//---------------------------------------------------------------------------------------------------------------
//
//  fb_Configuration
//
//  HAUD 2023.04.14
//  - base xml integration
//
//  HAUD 2026.04.10.
//  - now extending a base class
//
//  - cyclic OnChange wrapper for xml data 
//      - Ctrl/State
//        1. INIT
//        2. READ / WRITE
//
//  - read  ST_STATION_PARAMETER on demand
//  - write ST_STATION_PARAMETER on demand
//
//---------------------------------------------------------------------------------------------------------------
// This SOFTWARE is provided as an Example by THE PROVIDER "as is" and "with all faults." THE PROVIDER makes no 
// representations or warranties of any kind concerning the safety, suitability, lack of viruses, inaccuracies, 
// typographical errors, or other harmful components of this SOFTWARE. There are inherent dangers in the use of 
// any software, and you are solely responsible for determining whether this SOFTWARE is compatible with your 
// equipment and other software installed on your equipment. You are also solely responsible for the protection 
// of your equipment and backup of your data, and THE PROVIDER will not be liable for any damages you may suffer 
// in connection with using, modifying, or distributing this SOFTWARE.
//---------------------------------------------------------------------------------------------------------------
FUNCTION_BLOCK fb_Configuration EXTENDS fb_XmlBase
VAR
  _stCtrl               : REFERENCE TO ST_DATA_CTRL;
  _stState              : REFERENCE TO ST_DATA_STATE;

  _stConfiguration      : ST_Configuration;
  _pParameter           : POINTER TO ST_CONFIG_PORTAL;
END_VAR
VAR CONSTANT
  FILE_ROOT             : STRING := 'CONFIG_APPLICATION_';
  X_PATH                : STRING := '/config';
END_VAR

//---------------------------------------------------------------------------------------------------------------
//  check pointers from the outside
//---------------------------------------------------------------------------------------------------------------
IF NOT Check() THEN RETURN; END_IF
//---------------------------------------------------------------------------------------------------------------
// always build the internal data pointer
//  - as always: better safe than sorry
//  - leave this bit here, it doesn't cost much and safely addresses the data
//---------------------------------------------------------------------------------------------------------------
_pData                        := ADR    (_stConfiguration);
_nData                        := SIZEOF (_stConfiguration);
_sXpath                       := X_PATH;

// copy to local for debug
_eCmd                         := _stCtrl.Cmd;

// cyclic check for command change
// get state for cmd
IF (_eCmd <> _eCmdOld)
THEN
  // get matching sdtate for Ctrl.Cmd
  _eState                     := Cmd(_eCmd);
  _eCmdOld                    := _eCmd;
END_IF


CASE _eResult
OF
  E_PROGRESS.PROGRESS_INVALID:
    _stState.State            := E_DATA_STATE.NULL;

  E_PROGRESS.PROGRESS_ERROR:
    _stState.State            := _eState + E_PROGRESS.PROGRESS_ERROR;

  E_PROGRESS.PROGRESS_DONE:
    _stState.State            := _eState + E_PROGRESS.PROGRESS_DONE;

ELSE
  // work in progress
  // update progress for extern use
  _stState.State              := _eState + _eResult;

  CASE _eState
  OF
    E_DATA_STATE.INIT:
      _eResult   := _eInit    := CreateFolder(TRUE);

    E_DATA_STATE.READ:
      _eResult                := XmlRead(TRUE);
      IF (_eResult = E_PROGRESS.PROGRESS_DONE)
      THEN
        // copy the single ladies
        memcpy(_pParameter, ADR(_stConfiguration.PortalConfig), SIZEOF(_stConfiguration.PortalConfig));
      END_IF

    E_DATA_STATE.WRITE:
      _eResult                := XmlWrite(TRUE);
  ELSE
      _eResult                := E_PROGRESS.PROGRESS_INVALID;
  END_CASE
END_CASE

METHOD Check : BOOL
//-------------------------------------------------------------------------
IF NOT (__ISVALIDREF(_stCtrl))
THEN
  _eCheck               := E_DATA_CHECK.REFERENCE_CTRL_INVALID;
  RETURN;
END_IF
//-------------------------------------------------------------------------
IF NOT (__ISVALIDREF(_stState))
THEN
  _eCheck               := E_DATA_CHECK.REFERENCE_STATE_INVALID;
  RETURN;
END_IF
//-------------------------------------------------------------------------
IF NOT (_pStationParameter <> 0)
THEN
  _eCheck               := E_DATA_CHECK.POINTER_STATION_PARAMETER_INVALID;
  RETURN;
END_IF
//-------------------------------------------------------------------------
_eCheck                 := E_DATA_CHECK.DONE_CHECK;
Check                   := TRUE;
END_METHOD

METHOD PRIVATE Cmd : E_DATA_STATE
VAR_INPUT
  Ctrl      : E_DATA_CTRL;
END_VAR
VAR_INST
  _eState   : E_DATA_STATE;
END_VAR
IF NOT Check() THEN Cmd   := E_DATA_STATE.NULL;  RETURN; END_IF

CASE Ctrl
OF
  //---------------------------------------------------------------
  E_DATA_CTRL.INIT:
    _sName                := concat(FILE_ROOT, _sIdentity);
    _sName                := concat(_sName, '.xml');
    _sFilePath            := concat(_sDirectoryPath, _sName);

    _eInit                := E_PROGRESS.PROGRESS_INVALID;
    _eResult              := CreateFolder(FALSE);
    _eState               := E_DATA_STATE.INIT;
  //---------------------------------------------------------------
  E_DATA_CTRL.READ:
    _eResult              := XmlRead(FALSE);
    _eState               := E_DATA_STATE.READ;
  //---------------------------------------------------------------
  E_DATA_CTRL.WRITE:
    _stConfiguration.XtsStationParameter  := _pStationParameter^;

    _eResult              := XmlWrite(FALSE);
    _eState               := E_DATA_STATE.WRITE;
ELSE
  //---------------------------------------------------------------
    _eResult              := E_PROGRESS.PROGRESS_INVALID; 
    _eState               := E_DATA_STATE.NO_EXIST;
END_CASE

Cmd                       := _eState;
END_METHOD

PROPERTY Ctrl : REFERENCE to ST_DATA_CTRL
SET
_stCtrl ref= Ctrl;
END_SET
END_PROPERTY

PROPERTY Identity : OTCID
GET
Identity := _XpuIdentity;
END_GET
SET
_XpuIdentity  := Identity;
_sIdentity    := Tc2_Utilities.DWORD_TO_HEXSTR(_XpuIdentity,8,FALSE);
END_SET
END_PROPERTY

PROPERTY PortalConfig : POINTER TO ST_CONFIG_PORTAL
SET
_pParameter := PortalConfig;
END_SET
END_PROPERTY

PROPERTY State : REFERENCE TO ST_DATA_STATE
SET
_stState ref= State;
END_SET
END_PROPERTY

END_FUNCTION_BLOCK

(* stored: Version 1.1.0.1
   POU fb_Configuration: Id {35ac3f07-6ff4-42bc-88cc-d4fddf4268aa}, SpecialFunc None
   Folder methods: Id {1e2e40f2-6b00-45f7-a26e-c3cfe7d6b373}
   Folder properties: Id {da1a0b12-5642-438c-b8de-4af674c71976}
   Method Check: Id {43846077-1f15-499f-9f55-f39fe05d9613}
   Method Cmd: Id {f5160ffe-13d8-420d-82e9-9561109925e3}
   Property Ctrl: Id {9aa769b8-3546-48c2-a41b-d40a9aa36130}
   Set Set: Id {bc66070d-a937-4ae9-8da1-ab5d3c85346a}
   Property Identity: Id {9d072756-9a6f-436a-ae60-09f9df61e210}
   Get Get: Id {c0def124-ec06-4787-b726-86ab7ced8fa2}
   Set Set: Id {f5c2b1a3-2dde-46d1-af53-8529e98cfc59}
   Property PortalConfig: Id {4c83cfb6-f258-4f84-864e-c903031fb07c}
   Set Set: Id {d1e22c7d-f2eb-4b29-9846-670a06be153e}
   Property State: Id {c8aff51c-b2b8-43f2-9be9-db819b687773}
   Set Set: Id {d2e2f591-7465-4c7a-b025-49e9506ea3e6} *)
